{attribute addProperty BoxType "IODEVICETYPE_ETHERCATPROT"}
{attribute addProperty Id "TcTerminals210_2EK1100TcTerminals210_2EK1100_BDAFA3B600SyncUnitsSyncUnits_3FA29F3C21627InputsInputs_C75D3FEC1280160OutputsOutputs_47D1E803848106InfoDataInfoData_45F98C5022428"}
{attribute addProperty CRC "2929496954"}
{attribute addProperty SizeInBites "2568"}
{attribute addProperty SizeInBytes "321"}
TYPE EtherCAT_Master_KLxxxx_2_AE9C937A :
STRUCT
	{attribute addProperty Name "TcTerminals210_2EK1100"}
	TcTerminals210_2EK1100 : TcTerminals210_2EK1100_BDAFA3B6;
	{attribute addProperty Name "SyncUnits"}
	SyncUnits : SyncUnits_3FA29F3C;
	{attribute addProperty Name "Inputs"}
	Inputs : Inputs_C75D3FEC;
	{attribute addProperty Name "Outputs"}
	Outputs : Outputs_47D1E803;
	{attribute addProperty Name "InfoData"}
	InfoData : InfoData_45F98C50;
END_STRUCT
END_TYPE

(* stored: Version 1.2.0.0, ProductVersion 3.1.4024.9
   DUT EtherCAT_Master_KLxxxx_2_AE9C937A: Id {63d31b2a-73e2-496b-a6a8-dd3f9a7effa4} *)
